Fanuc KAREL source: ka00002.KL

PROGRAM KA00002
%NOLOCKGROUP
VAR
SRC:INTEGER;DST:REAL
BEGIN
--
SRC=2
DST=SRC
END KA00002
